Staubli VAL3: check_sphere.pgx

public program check_sphere(tool x_tTool, bool& x_bCheck[])
  local point l_pPoint
begin
  //
  // CHECK IF THE TOOL IS INSIDE
  //
  x_bCheck=false
  //
  if bCreate_sphere
    l_pPoint=here(x_tTool,world)
    // sphere
    if distance(pOrigin_sphere,l_pPoint)<=nRadius_sphere
      // check if inside
      x_bCheck=true
    endIf
  endIf
end
